% RSLogix 500 project rev_pulse.RSS, saved by version 8.30.00.16 %
PROJECT "UNTITLED"    % processor: Bul.1763 MicroLogix 1100 Series B %

PROGRAM FILES
  LAD 2   5 rungs

DATA FILES
  O0 OUTPUT  4 elements
  I1 INPUT  6 elements
  S2 STATUS  66 elements
  B3 BINARY  24 elements
  T4 TIMER  1 elements
  C5 COUNTER  1 elements
  R6 CONTROL  1 elements
  N7 INTEGER  52 elements
  F8 FLOAT  1 elements
  C15   1 elements
  F18   11 elements
  L20 LONG MATH  10 elements

LADDER 2
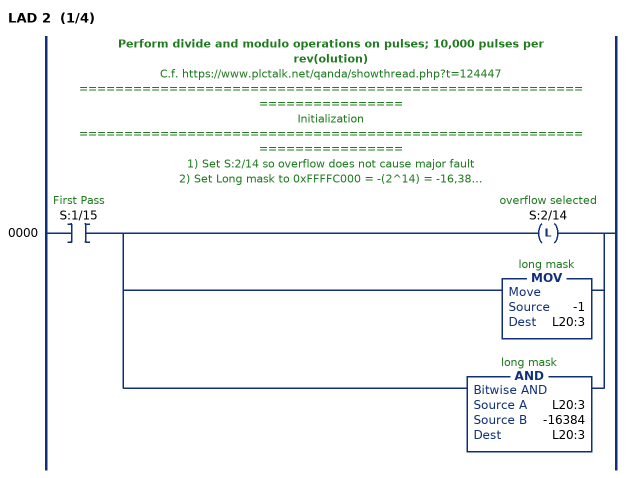
% Rung: 0 %
% TITLE: Perform divide and modulo operations on pulses; 10,000 pulses per rev(olution) %
% C.f. https://www.plctalk.net/qanda/showthread.php?t=124447
% 
% 
% ========================================================================
% Initialization
% ========================================================================
% 
% 1) Set S:2/14 so overflow does not cause major fault
% 
% 2) Set Long mask to 0xFFFFC000 = -(2^14) = -16,384
% 2.1) Use MOV -1 (0xFFFFFFFF) and AND so mask will be seen in hex %
SOR XIC S:1/15 BST OTL S:2/14 NXB MOV -1 L20:3 NXB AND L20:3 -16384 L20:3 BND EOR
%   S:1/15  "First Pass" %
%   S:2/14  "overflow selected" %
%   L20:3  "long mask" %

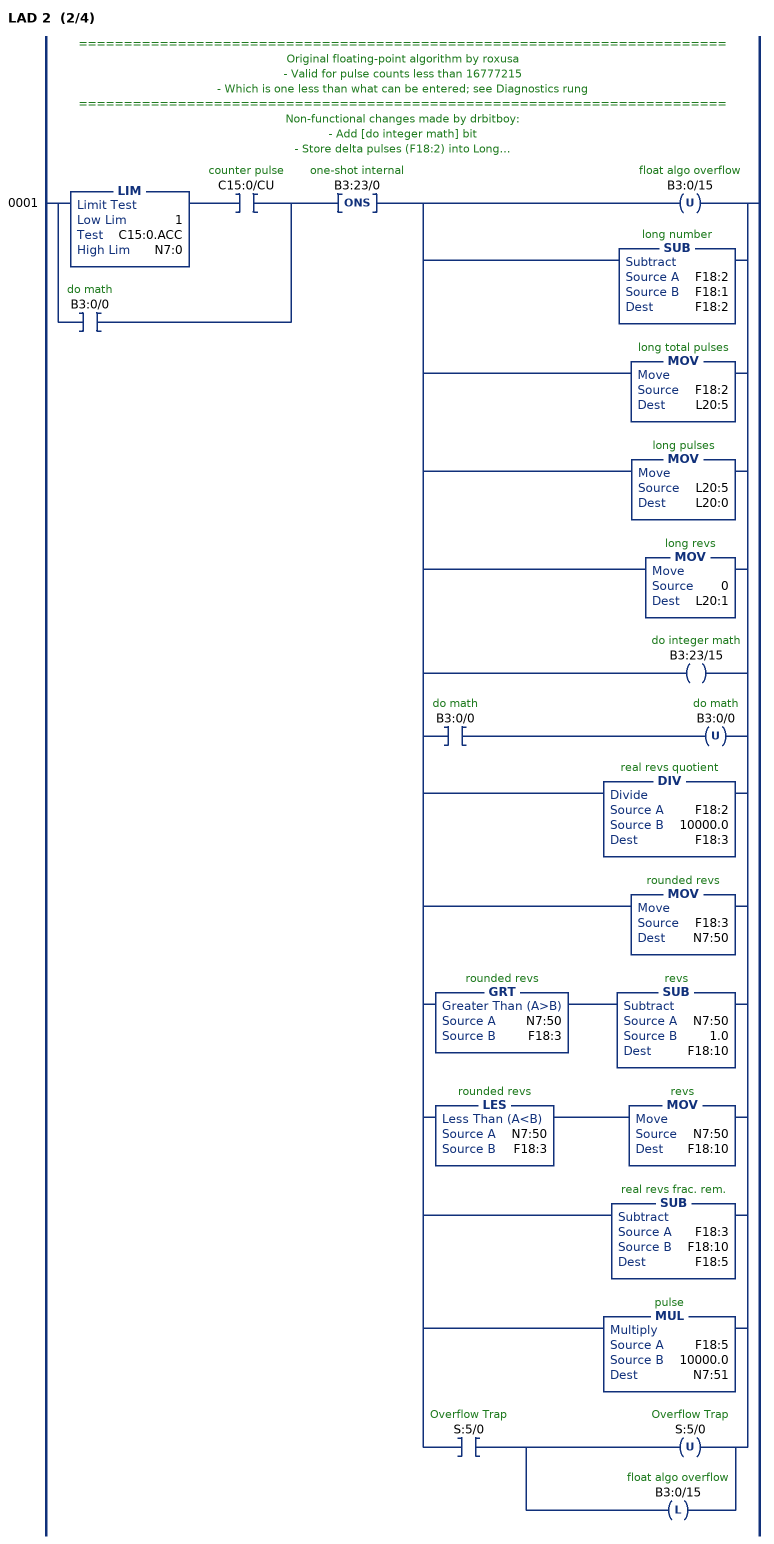
% Rung: 1 %
% ========================================================================
% Original floating-point algorithm by roxusa
% - Valid for pulse counts less than 16777215
%   - Which is one less than what can be entered; see Diagnostics rung
% ========================================================================
% Non-functional changes made by drbitboy:
% 
% - Add [do integer math] bit
% - Store delta pulses (F18:2) into Longs
% - Clear manual [do math] bit
% - Clear any overflow at end of rung %
SOR BST LIM 1 C15:0.ACC N7:0 XIC C15:0/CU NXB XIC B3:0/0 BND ONS B3:23/0 BST OTU B3:0/15 NXB SUB F18:2 F18:1 F18:2 NXB BST MOV F18:2 L20:5 NXB MOV L20:5 L20:0 NXB MOV 0 L20:1 NXB OTE B3:23/15 NXB XIC B3:0/0 OTU B3:0/0 BND NXB DIV F18:2 10000.0 F18:3 NXB MOV F18:3 N7:50 NXB GRT N7:50 F18:3 SUB N7:50 1.0 F18:10 NXB LES N7:50 F18:3 MOV N7:50 F18:10 NXB SUB F18:3 F18:10 F18:5 NXB MUL F18:5 10000.0 N7:51 NXB XIC S:5/0 BST OTU S:5/0 NXB OTL B3:0/15 BND BND EOR
%   N7:0  "Bundle Preset" %
%   C15:0/CU  "counter pulse" %
%   B3:0/0  "do math" %
%   B3:23/0  "one-shot internal" %
%   B3:0/15  "float algo overflow" %
%   F18:2  "long number" %
%   F18:1  "drop amount" %
%   L20:5  "long total pulses" %
%   L20:0  "long pulses" %
%   L20:1  "long revs" %
%   B3:23/15  "do integer math" %
%   F18:3  "real revs quotient" %
%   N7:50  "rounded revs" %
%   F18:10  "revs" %
%   F18:5  "real revs frac. rem." %
%   N7:51  "pulse" %
%   S:5/0  "Overflow Trap" %

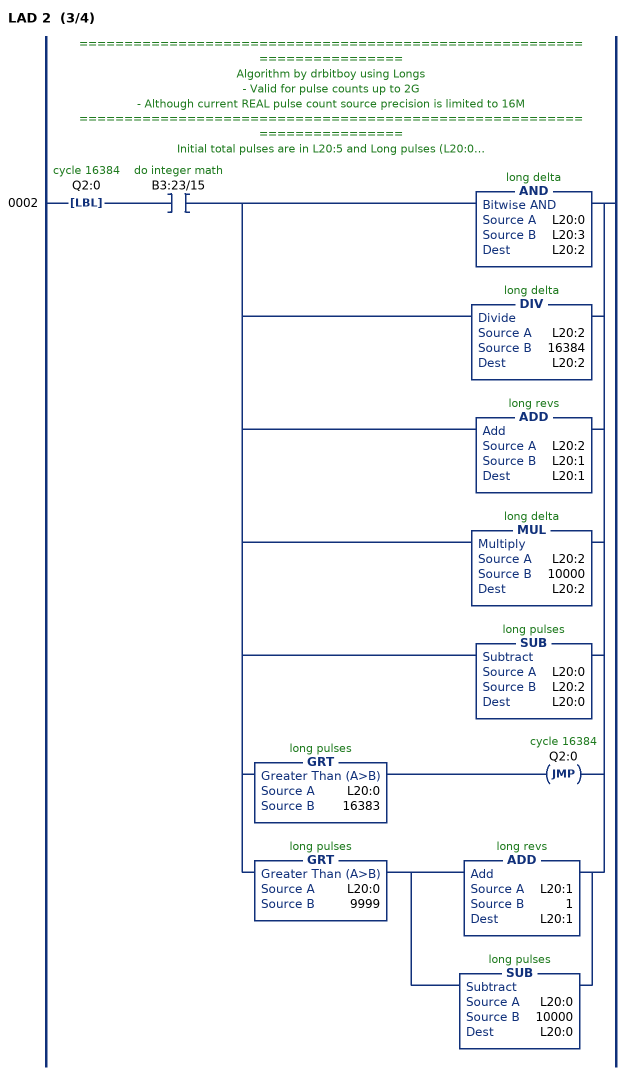
% Rung: 2 %
% ========================================================================
% Algorithm by drbitboy using Longs
% - Valid for pulse counts up to 2G
%   - Although current REAL pulse count source precision is limited to 16M
% ========================================================================
% Initial total pulses are in L20:5 and Long pulses (L20:0)
% - Moved from F18:2 in rung 0001 above
% 
% Summary
% - Long pulses will be reduced to the remaining pulses = L20:5 MODULO 10000
% - Long revs (L 20:1) will contain the number of 10kpulse revs
% 
% Implementation details
% - Loop
%   - Get truncated quotient Long delta = (Long pulses) / 16384
%   - Add Long delta to Long revs (L20:1)
%   - Subtract (10000 * (Long delta)) from Long pulses
%   - Repeat loop as long as (Long pulses) valule is greater than 16383,
% - After looping is complete, if Long pulses value is greater than 9999
%   - Add 1 to revs
%   - Subtract 10000 from Long pulses %
SOR LBL Q2:0 XIC B3:23/15 BST AND L20:0 L20:3 L20:2 NXB DIV L20:2 16384 L20:2 NXB ADD L20:2 L20:1 L20:1 NXB MUL L20:2 10000 L20:2 NXB SUB L20:0 L20:2 L20:0 NXB GRT L20:0 16383 JMP Q2:0 NXB GRT L20:0 9999 BST ADD L20:1 1 L20:1 NXB SUB L20:0 10000 L20:0 BND BND EOR
%   Q2:0  "cycle 16384" %
%   B3:23/15  "do integer math" %
%   L20:0  "long pulses" %
%   L20:3  "long mask" %
%   L20:2  "long delta" %
%   L20:1  "long revs" %

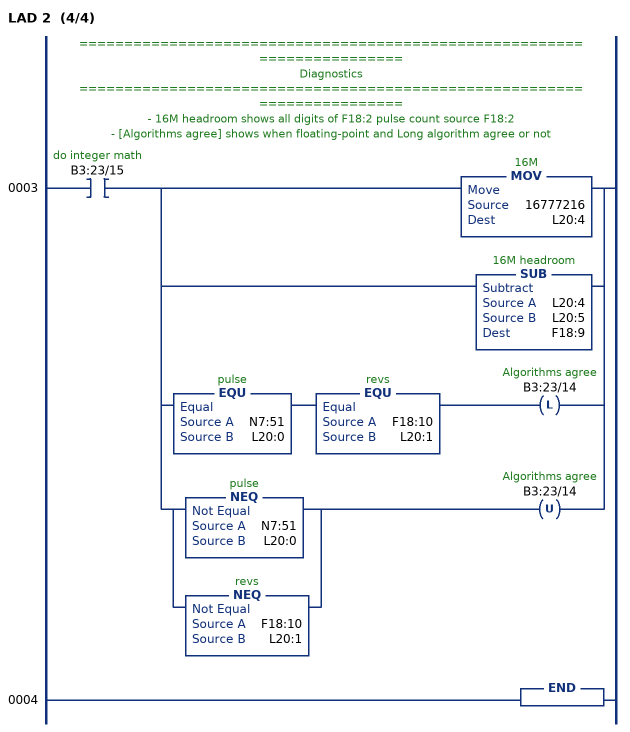
% Rung: 3 %
% ========================================================================
% Diagnostics
% ========================================================================
% - 16M headroom shows all digits of F18:2 pulse count source F18:2
% - [Algorithms agree] shows when floating-point and Long algorithm agree or not %
SOR XIC B3:23/15 BST MOV 16777216 L20:4 NXB SUB L20:4 L20:5 F18:9 NXB EQU N7:51 L20:0 EQU F18:10 L20:1 OTL B3:23/14 NXB BST NEQ N7:51 L20:0 NXB NEQ F18:10 L20:1 BND OTU B3:23/14 BND EOR
%   B3:23/15  "do integer math" %
%   L20:4  "16M" %
%   L20:5  "long total pulses" %
%   F18:9  "16M headroom" %
%   N7:51  "pulse" %
%   L20:0  "long pulses" %
%   F18:10  "revs" %
%   L20:1  "long revs" %
%   B3:23/14  "Algorithms agree" %
% Rung: 4 %
SOR END EOR
